// TIA Portal V17 export
// export: Created 2025-06-26T06:49:19.1246133Z, ExportSetting WithDefaults, DisplayName Totally Integrated Automation Portal, DisplayVersion V17 Update 8, DisplayName TIA Portal Openness, DisplayVersion V17 Update 8, DisplayName TIA Portal Version Control Interface, DisplayVersion V17, DisplayName STEP 7 Professional, DisplayVersion V17 Update 8, DisplayName STEP 7 Safety, DisplayVersion V17 Update 6, DisplayName WinCC Advanced, DisplayVersion V17 Update 8
FUNCTION "AnalogOutputProcessing" : Void   // FC12, FBD
TITLE = Output mapping and scaling
{ S7_Optimized_Access := 'TRUE' }
VERSION : 0.1
// stored: AutoNumber true, IsIECCheckEnabled false, SetENOAutomatically false, UDAEnableTagReadback false
BEGIN

REGION Network 1: HBL-HCV-576
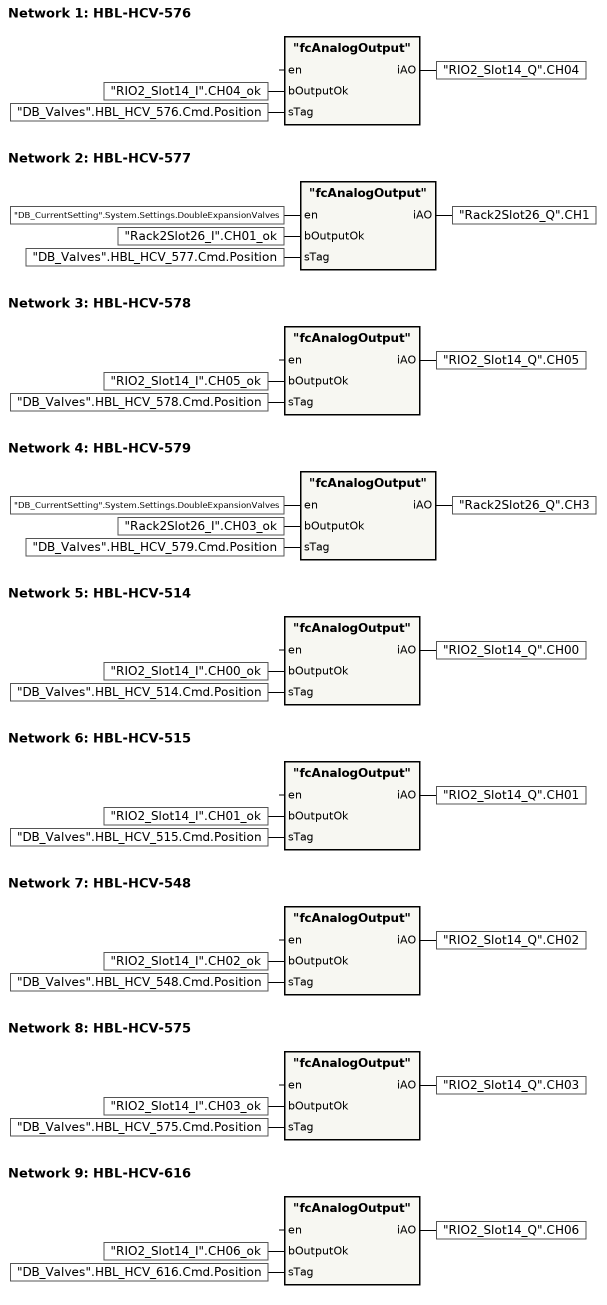
   "fcAnalogOutput"(bOutputOk := "RIO2_Slot14_I".CH04_ok,
                    sTag := "DB_Valves".HBL_HCV_576.Cmd.Position,
                    iAO => "RIO2_Slot14_Q".CH04);
END_REGION

REGION Network 2: HBL-HCV-577
   IF "DB_CurrentSetting".System.Settings.DoubleExpansionValves THEN
       "fcAnalogOutput"(bOutputOk := "Rack2Slot26_I".CH01_ok,
                        sTag := "DB_Valves".HBL_HCV_577.Cmd.Position,
                        iAO => "Rack2Slot26_Q".CH1);
   END_IF;
END_REGION

REGION Network 3: HBL-HCV-578
   "fcAnalogOutput"(bOutputOk := "RIO2_Slot14_I".CH05_ok,
                    sTag := "DB_Valves".HBL_HCV_578.Cmd.Position,
                    iAO => "RIO2_Slot14_Q".CH05);
END_REGION

REGION Network 4: HBL-HCV-579
   IF "DB_CurrentSetting".System.Settings.DoubleExpansionValves THEN
       "fcAnalogOutput"(bOutputOk := "Rack2Slot26_I".CH03_ok,
                        sTag := "DB_Valves".HBL_HCV_579.Cmd.Position,
                        iAO => "Rack2Slot26_Q".CH3);
   END_IF;
END_REGION

REGION Network 5: HBL-HCV-514
   "fcAnalogOutput"(bOutputOk := "RIO2_Slot14_I".CH00_ok,
                    sTag := "DB_Valves".HBL_HCV_514.Cmd.Position,
                    iAO => "RIO2_Slot14_Q".CH00);
END_REGION

REGION Network 6: HBL-HCV-515
   "fcAnalogOutput"(bOutputOk := "RIO2_Slot14_I".CH01_ok,
                    sTag := "DB_Valves".HBL_HCV_515.Cmd.Position,
                    iAO => "RIO2_Slot14_Q".CH01);
END_REGION

REGION Network 7: HBL-HCV-548
   "fcAnalogOutput"(bOutputOk := "RIO2_Slot14_I".CH02_ok,
                    sTag := "DB_Valves".HBL_HCV_548.Cmd.Position,
                    iAO => "RIO2_Slot14_Q".CH02);
END_REGION

REGION Network 8: HBL-HCV-575
   "fcAnalogOutput"(bOutputOk := "RIO2_Slot14_I".CH03_ok,
                    sTag := "DB_Valves".HBL_HCV_575.Cmd.Position,
                    iAO => "RIO2_Slot14_Q".CH03);
END_REGION

REGION Network 9: HBL-HCV-616
   "fcAnalogOutput"(bOutputOk := "RIO2_Slot14_I".CH06_ok,
                    sTag := "DB_Valves".HBL_HCV_616.Cmd.Position,
                    iAO => "RIO2_Slot14_Q".CH06);
END_REGION

REGION Network 10: HBL-HCV-700
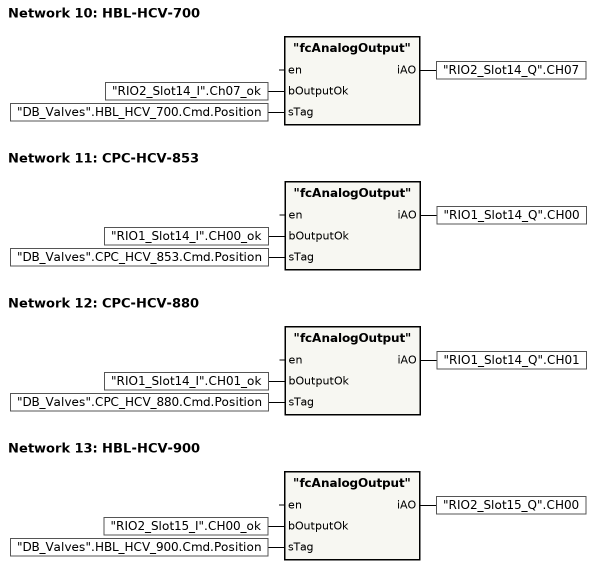
   "fcAnalogOutput"(bOutputOk := "RIO2_Slot14_I".Ch07_ok,
                    sTag := "DB_Valves".HBL_HCV_700.Cmd.Position,
                    iAO => "RIO2_Slot14_Q".CH07);
END_REGION

REGION Network 11: CPC-HCV-853
   "fcAnalogOutput"(bOutputOk := "RIO1_Slot14_I".CH00_ok,
                    sTag := "DB_Valves".CPC_HCV_853.Cmd.Position,
                    iAO => "RIO1_Slot14_Q".CH00);
END_REGION

REGION Network 12: CPC-HCV-880
   "fcAnalogOutput"(bOutputOk := "RIO1_Slot14_I".CH01_ok,
                    sTag := "DB_Valves".CPC_HCV_880.Cmd.Position,
                    iAO => "RIO1_Slot14_Q".CH01);
END_REGION

REGION Network 13: HBL-HCV-900
   "fcAnalogOutput"(bOutputOk := "RIO2_Slot15_I".CH00_ok,
                    sTag := "DB_Valves".HBL_HCV_900.Cmd.Position,
                    iAO => "RIO2_Slot15_Q".CH00);
END_REGION
END_FUNCTION
